FUNCTION_BLOCK FB_AxisGroups
VAR_INPUT
END_VAR
VAR_OUTPUT
END_VAR
VAR
	_stAxisGroup: REFERENCE TO ST_AxisGroupStruct;
	iGroupedAxis : INT;
END_VAR

METHOD mStatus_GroupEnabled : BOOL
VAR_INPUT
END_VAR
_stAxisGroup.stFlag.iDisabled := 0;
_stAxisGroup.stFlag.bDisabledFlag := FALSE;
_stAxisGroup.stFlag.iNumberOfAxisDisabled := 0;
FOR iGroupedAxis := 1 TO GVL.nMAX_AXES_PER_GROUP DO
	IF _stAxisGroup.aAxesInGroup[iGroupedAxis] = 0 THEN
		IF _stAxisGroup.stFlag.iDisabled <> 0 THEN
			_stAxisGroup.stFlag.bDisabledFlag := TRUE;	
		END_IF
		RETURN;
	END_IF
	_stAxisGroup.stFlag.iDisabled := _stAxisGroup.stFlag.iDisabled + BOOL_TO_INT(NOT astAxes[_stAxisGroup.aAxesInGroup[iGroupedAxis]].stStatus.bEnabled) * iGroupedAxis;
	_stAxisGroup.stFlag.iNumberOfAxisDisabled := _stAxisGroup.stFlag.iNumberOfAxisDisabled + BOOL_TO_INT(NOT astAxes[_stAxisGroup.aAxesInGroup[iGroupedAxis]].stStatus.bEnabled);
END_FOR
END_METHOD

METHOD mStatus_GroupError : BOOL
VAR_INPUT
END_VAR
_stAxisGroup.stFlag.iError := 0;
_stAxisGroup.stFlag.bErrorFlag := FALSE;
_stAxisGroup.stFlag.iNumberOfAxisInError := 0; 

FOR iGroupedAxis := 1 TO GVL.nMAX_AXES_PER_GROUP DO
	IF _stAxisGroup.aAxesInGroup[iGroupedAxis] = 0 THEN
		IF _stAxisGroup.stFlag.iError <> 0 THEN
			_stAxisGroup.stFlag.bErrorFlag := TRUE;
		END_IF
		RETURN;
	END_IF
	_stAxisGroup.stFlag.iError := _stAxisGroup.stFlag.iError + BOOL_TO_INT(astAxes[_stAxisGroup.aAxesInGroup[iGroupedAxis]].stStatus.bError) * (100 + iGroupedAxis);
	_stAxisGroup.stFlag.iNumberOfAxisInError := _stAxisGroup.stFlag.iNumberOfAxisInError + BOOL_TO_INT(astAxes[_stAxisGroup.aAxesInGroup[iGroupedAxis]].stStatus.bError);
END_FOR
END_METHOD

METHOD mStatus_GroupState : BOOL
VAR_INPUT
END_VAR
_stAxisGroup.stFlag.iState := _stAxisGroup.stFlag.iDisabled + _stAxisGroup.stFlag.iError;
END_METHOD

METHOD Run : BOOL
VAR_INPUT
END_VAR
mStatus_GroupEnabled();
mStatus_GroupError();
mStatus_GroupState();
END_METHOD

PROPERTY stAxisGroup : REFERENCE TO ST_AxisGroupStruct
GET
stAxisGroup REF= _stAxisGroup;
END_GET
SET
_stAxisGroup REF= stAxisGroup;
END_SET
END_PROPERTY

END_FUNCTION_BLOCK

(* stored: Version 1.1.0.1, ProductVersion 3.1.4024.11
   POU FB_AxisGroups: Id {3d34cf0c-94a1-435c-a681-8b8d3300efd6}, SpecialFunc None
   Method mStatus_GroupEnabled: Id {6497340e-04cd-4c6c-b84a-9262b3cfb20a}
   Method mStatus_GroupError: Id {fee155b1-4d8e-4a2a-af48-41dce12c5c37}
   Method mStatus_GroupState: Id {ac5aa7c0-cdbe-4a70-9534-676d39efbaa7}
   Method Run: Id {1f8f2b5c-38ba-47df-a074-81ee7eecc5fd}
   Property stAxisGroup: Id {09889def-20eb-4fe2-9b02-3e045fae4d3b}
   Get Get: Id {c34f8397-af38-407f-8435-195eb63bbcfc}
   Set Set: Id {07562d57-b69c-4492-b5f7-7067c20a4c32} *)
